VAR_GLOBAL CONSTANT
    cTimeout : TIME := T#5S;
END_VAR
VAR_GLOBAL RETAIN
    nBootCount : UDINT;
END_VAR

(* stored: Version 1.1.0.1, ProductVersion 3.1.4024.16
   GVL GVL_Syntax_Global: Id {f85e7ddd-6af3-415f-b7ca-7d94f9a52f74} *)
